TYPE ST_HMI_COLOR_STRING : STRUCT
	color: STRING; (* Defining a color as CSS color: #hexadecimal, rgb(), rgba(), hsl(), hsla(), css color keyword, none or transparent. *)
END_STRUCT
END_TYPE

(* stored: Version 1.1.0.1, ProductVersion 3.1.4024.11
   DUT ST_HMI_COLOR_STRING: Id {c10d9f8c-22ec-4572-9154-0ef977f37120} *)
